(* LS Electric XG5000 project: 241008_연습문제11 *)
(* PLC LSPLC *)

PROGRAM NewProgram (* task: 스캔 프로그램 *)
VAR
    P1 AT %IX0.0.1 : BOOL;
    P10 AT %QX0.1.0 : BOOL;
    P11 AT %QX0.1.1 : BOOL;
    PUSH AT %IX0.0.0 : BOOL;
    T1 : CTU_INT;
    T2 : CTU_INT;
    T3 : CTU_INT;
END_VAR

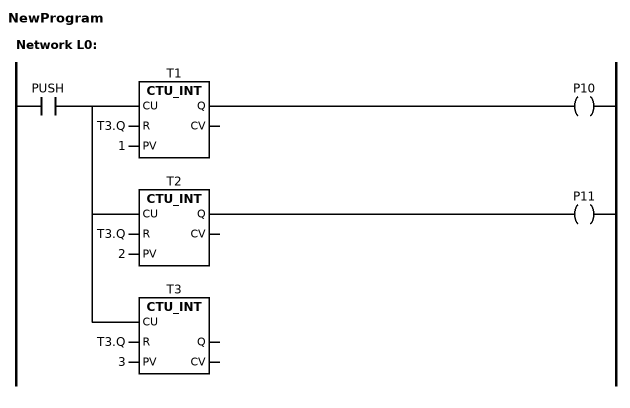
(* Rung L0 *)
T1(CU := PUSH, R := T3.Q, PV := 1);
P10 := T1.Q;
T2(CU := PUSH, R := T3.Q, PV := 2);
P11 := T2.Q;
T3(CU := PUSH, R := T3.Q, PV := 3);
END_PROGRAM